// TIA Portal V20 export
TYPE "LPFE_typeAlarmClassifications"
// stored: Access Published, Namespace PFE
   STRUCT
      Fault { S7_SetPoint := 'True'} : "PFE.LPFE_typeFault";
      Warning { S7_SetPoint := 'True'} : "PFE.LPFE_typeWarning";
      Status { S7_SetPoint := 'True'} : "PFE.LPFE_typeStatus";
   END_STRUCT;
END_TYPE
